# EPICS substitutions: ek9000App/Db/EL3161.substitutions
file EL3161.template
{       pattern
        {
                TERMINAL,

        }
        {
        }
}
